INTERFACE ITF_SaMControllerCommandChange

METHOD PUBLIC ChangeStateBusy : BOOL
VAR_INPUT
END_VAR
END_METHOD

METHOD PUBLIC ChangeStateDone : BOOL
VAR_INPUT
END_VAR
END_METHOD

METHOD PUBLIC ChangeStateExecute : BOOL
VAR_INPUT
	eNewState			: E_SaMStates;
END_VAR
END_METHOD

END_INTERFACE

(* stored: Version 1.1.0.1
   Itf ITF_SaMControllerCommandChange: Id {4f3c20a9-bad8-0c25-32a4-4d92805aad72}
   Method ChangeStateBusy: Id {bcebd3f8-de4d-0c8f-1c39-4aa70f756c8f}
   Method ChangeStateDone: Id {5d2b48c0-ca69-0156-247c-adcdae5d65b3}
   Method ChangeStateExecute: Id {049dd90b-20e0-0046-1339-9d6e6a3dbad6} *)
